TYPE ST_LS_CfgLiftEncoder :
STRUCT
	Positions	: ST_LSPM_LiftEncPos;		// Encoder position configuration
	Preset		: ST_LS_CfgLiftEncPreset;	// Preset encoder information
END_STRUCT
END_TYPE

(* stored: Version 1.1.0.1, ProductVersion 3.1.4024.4
   DUT ST_LS_CfgLiftEncoder: Id {9d2a12b5-bfe0-4ae9-bb79-887b2ef91523} *)
